// TIA Portal V20 export
FUNCTION "CollectAlarms" : Void   // FC64, LAD
TITLE = Alarm Collector Unit
AUTHOR : ERsystem_FA2_DH. Kim
// Collects alarms from the respective level and categorises the alarms into the different alarm classes.
// stored: Namespace Unit1, SetENOAutomatically false
   VAR_INPUT
      resetAlarms : Bool;
      disableAlarms : Bool;
   END_VAR
   VAR_OUTPUT
      commandsToUnit : "LUC_typeStateCommands";   // Feedback to the unit
   END_VAR
   VAR CONSTANT
      DelayTime : Time := T#300ms;
      TRUE : Bool := TRUE;
      FALSE : Bool;
   END_VAR
BEGIN

REGION Network 1: Reset Alarms
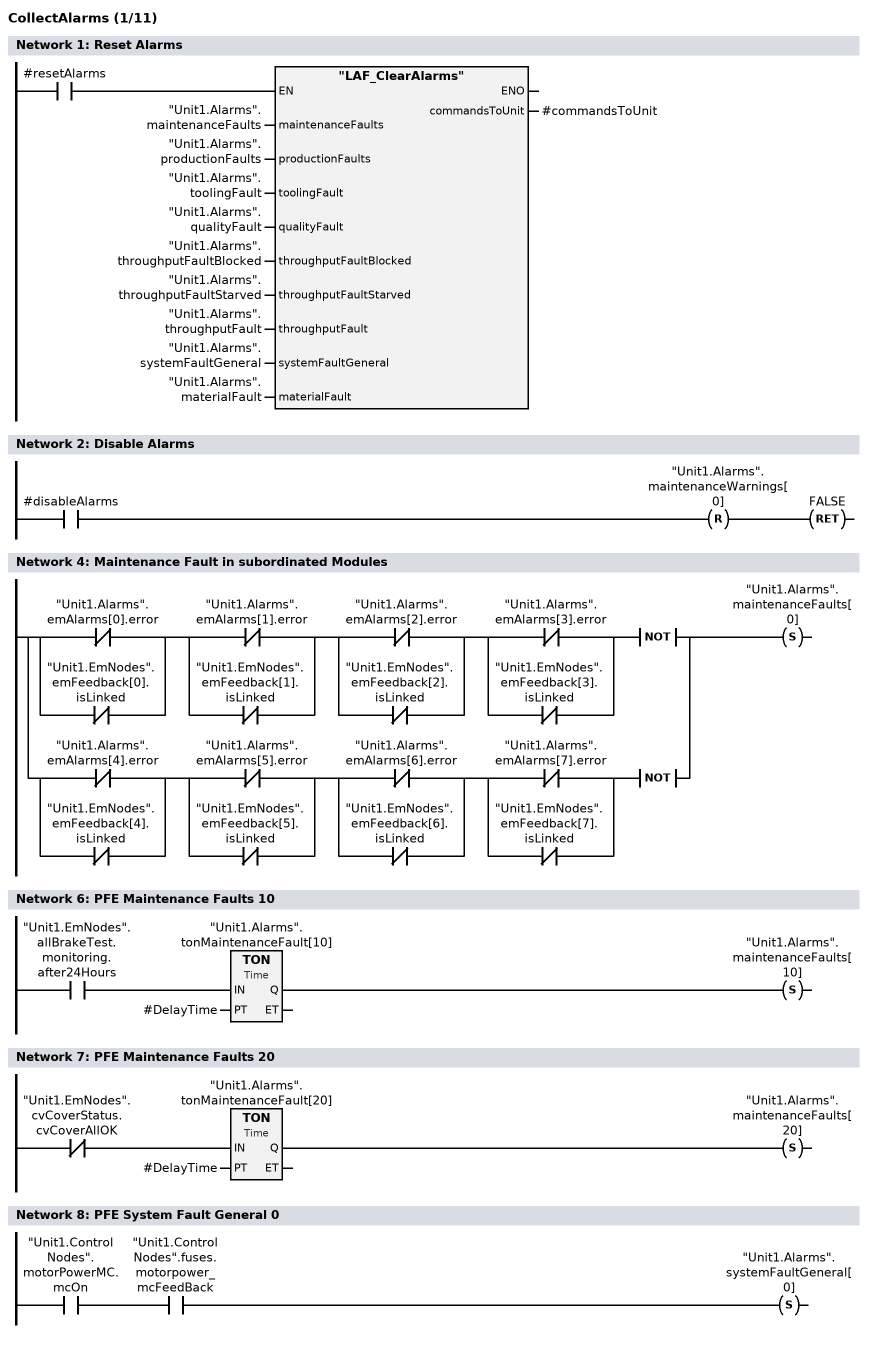
   RUNG wire#powerrail
      Contact( #resetAlarms )
      "LAF_ClearAlarms"(maintenanceFaults := "Unit1.Alarms".maintenanceFaults, productionFaults := "Unit1.Alarms".productionFaults, toolingFault := "Unit1.Alarms".toolingFault, qualityFault := "Unit1.Alarms".qualityFault, throughputFaultBlocked := "Unit1.Alarms".throughputFaultBlocked, throughputFaultStarved := "Unit1.Alarms".throughputFaultStarved, throughputFault := "Unit1.Alarms".throughputFault, systemFaultGeneral := "Unit1.Alarms".systemFaultGeneral, materialFault := "Unit1.Alarms".materialFault, commandsToUnit => #commandsToUnit)
   END_RUNG
   // the same network as SCL:
   IF #resetAlarms THEN
       "LAF_ClearAlarms"(maintenanceFaults := "Unit1.Alarms".maintenanceFaults,
                         productionFaults := "Unit1.Alarms".productionFaults,
                         toolingFault := "Unit1.Alarms".toolingFault,
                         qualityFault := "Unit1.Alarms".qualityFault,
                         throughputFaultBlocked := "Unit1.Alarms".throughputFaultBlocked,
                         throughputFaultStarved := "Unit1.Alarms".throughputFaultStarved,
                         throughputFault := "Unit1.Alarms".throughputFault,
                         systemFaultGeneral := "Unit1.Alarms".systemFaultGeneral,
                         materialFault := "Unit1.Alarms".materialFault,
                         commandsToUnit => #commandsToUnit);
   END_IF;
END_REGION

REGION Network 2: Disable Alarms
   RUNG wire#powerrail
      Contact( #disableAlarms )
      R_Coil( "Unit1.Alarms".maintenanceWarnings[0] )
      ReturnCoil( FALSE )
   END_RUNG
   // the same network as SCL:
   IF #disableAlarms THEN
       "Unit1.Alarms".maintenanceWarnings[0] := FALSE;
       ENO := FALSE;
       RETURN;
   END_IF;
END_REGION

REGION Network 3: *************** Fault ************************
END_REGION

REGION Network 4: Maintenance Fault in subordinated Modules
   RUNG wire#powerrail
      I_Contact( "Unit1.Alarms".emAlarms[0].error )
      wire#w1
      I_Contact( "Unit1.Alarms".emAlarms[1].error )
      wire#w2
      I_Contact( "Unit1.Alarms".emAlarms[2].error )
      wire#w3
      I_Contact( "Unit1.Alarms".emAlarms[3].error )
      wire#w4
      Not()
      wire#w5
      S_Coil( "Unit1.Alarms".maintenanceFaults[0] )
   END_RUNG
   RUNG wire#powerrail
      I_Contact( "Unit1.EmNodes".emFeedback[0].isLinked )
   END_RUNG wire#w1
   RUNG wire#w1
      I_Contact( "Unit1.EmNodes".emFeedback[1].isLinked )
   END_RUNG wire#w2
   RUNG wire#w2
      I_Contact( "Unit1.EmNodes".emFeedback[2].isLinked )
   END_RUNG wire#w3
   RUNG wire#w3
      I_Contact( "Unit1.EmNodes".emFeedback[3].isLinked )
   END_RUNG wire#w4
   RUNG wire#powerrail
      I_Contact( "Unit1.Alarms".emAlarms[4].error )
      wire#w6
      I_Contact( "Unit1.Alarms".emAlarms[5].error )
      wire#w7
      I_Contact( "Unit1.Alarms".emAlarms[6].error )
      wire#w8
      I_Contact( "Unit1.Alarms".emAlarms[7].error )
      wire#w9
      Not()
   END_RUNG wire#w5
   RUNG wire#powerrail
      I_Contact( "Unit1.EmNodes".emFeedback[4].isLinked )
   END_RUNG wire#w6
   RUNG wire#w6
      I_Contact( "Unit1.EmNodes".emFeedback[5].isLinked )
   END_RUNG wire#w7
   RUNG wire#w7
      I_Contact( "Unit1.EmNodes".emFeedback[6].isLinked )
   END_RUNG wire#w8
   RUNG wire#w8
      I_Contact( "Unit1.EmNodes".emFeedback[7].isLinked )
   END_RUNG wire#w9
   // the same network as SCL:
   IF NOT ((NOT "Unit1.Alarms".emAlarms[0].error OR NOT "Unit1.EmNodes".emFeedback[0].isLinked) AND (NOT "Unit1.Alarms".emAlarms[1].error OR NOT "Unit1.EmNodes".emFeedback[1].isLinked) AND (NOT "Unit1.Alarms".emAlarms[2].error OR NOT "Unit1.EmNodes".emFeedback[2].isLinked) AND (NOT "Unit1.Alarms".emAlarms[3].error OR NOT "Unit1.EmNodes".emFeedback[3].isLinked)) OR NOT ((NOT "Unit1.Alarms".emAlarms[4].error OR NOT "Unit1.EmNodes".emFeedback[4].isLinked) AND (NOT "Unit1.Alarms".emAlarms[5].error OR NOT "Unit1.EmNodes".emFeedback[5].isLinked) AND (NOT "Unit1.Alarms".emAlarms[6].error OR NOT "Unit1.EmNodes".emFeedback[6].isLinked) AND (NOT "Unit1.Alarms".emAlarms[7].error OR NOT "Unit1.EmNodes".emFeedback[7].isLinked)) THEN
       "Unit1.Alarms".maintenanceFaults[0] := TRUE;
   END_IF;
END_REGION

REGION Network 5: PFE Maintenance Faults 1
END_REGION

REGION Network 6: PFE Maintenance Faults 10
   RUNG wire#powerrail
      Contact( "Unit1.EmNodes".allBrakeTest.monitoring.after24Hours )
      { S7_Templates := "time_type := Time" } "Unit1.Alarms".tonMaintenanceFault[10].TON(pt := #DelayTime, et =>)
      S_Coil( "Unit1.Alarms".maintenanceFaults[10] )
   END_RUNG
   // the same network as SCL:
   "Unit1.Alarms".tonMaintenanceFault[10].TON(IN := "Unit1.EmNodes".allBrakeTest.monitoring.after24Hours,
                           PT := #DelayTime);
   IF "Unit1.Alarms".tonMaintenanceFault[10].Q THEN "Unit1.Alarms".maintenanceFaults[10] := TRUE; END_IF;
END_REGION

REGION Network 7: PFE Maintenance Faults 20
   RUNG wire#powerrail
      I_Contact( "Unit1.EmNodes".cvCoverStatus.cvCoverAllOK )
      { S7_Templates := "time_type := Time" } "Unit1.Alarms".tonMaintenanceFault[20].TON(pt := #DelayTime, et =>)
      S_Coil( "Unit1.Alarms".maintenanceFaults[20] )
   END_RUNG
   // the same network as SCL:
   "Unit1.Alarms".tonMaintenanceFault[20].TON(IN := NOT "Unit1.EmNodes".cvCoverStatus.cvCoverAllOK,
                           PT := #DelayTime);
   IF "Unit1.Alarms".tonMaintenanceFault[20].Q THEN "Unit1.Alarms".maintenanceFaults[20] := TRUE; END_IF;
END_REGION

REGION Network 8: PFE System Fault General 0
   RUNG wire#powerrail
      Contact( "Unit1.ControlNodes".motorPowerMC.mcOn )
      Contact( "Unit1.ControlNodes".fuses.motorpower_mcFeedBack )
      S_Coil( "Unit1.Alarms".systemFaultGeneral[0] )
   END_RUNG
   // the same network as SCL:
   IF "Unit1.ControlNodes".motorPowerMC.mcOn AND "Unit1.ControlNodes".fuses.motorpower_mcFeedBack THEN
       "Unit1.Alarms".systemFaultGeneral[0] := TRUE;
   END_IF;
END_REGION

REGION Network 9: PFE System Fault General 1
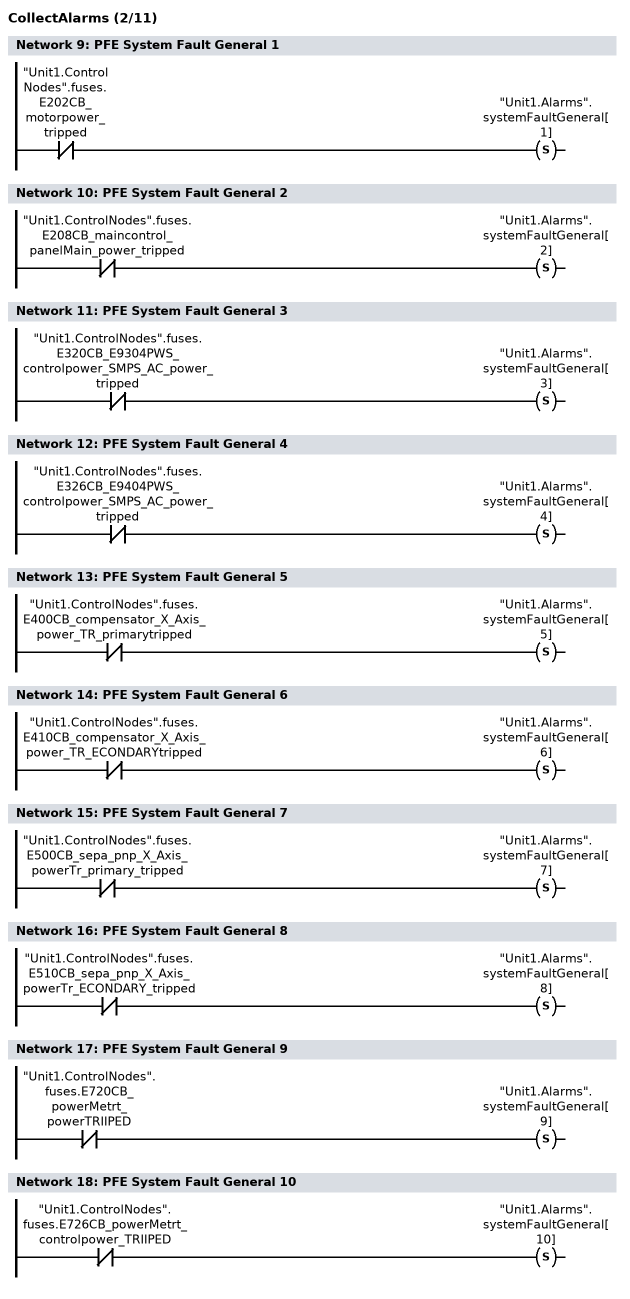
   RUNG wire#powerrail
      I_Contact( "Unit1.ControlNodes".fuses.E202CB_motorpower_tripped )
      S_Coil( "Unit1.Alarms".systemFaultGeneral[1] )
   END_RUNG
   // the same network as SCL:
   IF NOT "Unit1.ControlNodes".fuses.E202CB_motorpower_tripped THEN
       "Unit1.Alarms".systemFaultGeneral[1] := TRUE;
   END_IF;
END_REGION

REGION Network 10: PFE System Fault General 2
   RUNG wire#powerrail
      I_Contact( "Unit1.ControlNodes".fuses.E208CB_maincontrol_panelMain_power_tripped )
      S_Coil( "Unit1.Alarms".systemFaultGeneral[2] )
   END_RUNG
   // the same network as SCL:
   IF NOT "Unit1.ControlNodes".fuses.E208CB_maincontrol_panelMain_power_tripped THEN
       "Unit1.Alarms".systemFaultGeneral[2] := TRUE;
   END_IF;
END_REGION

REGION Network 11: PFE System Fault General 3
   RUNG wire#powerrail
      I_Contact( "Unit1.ControlNodes".fuses.E320CB_E9304PWS_controlpower_SMPS_AC_power_tripped )
      S_Coil( "Unit1.Alarms".systemFaultGeneral[3] )
   END_RUNG
   // the same network as SCL:
   IF NOT "Unit1.ControlNodes".fuses.E320CB_E9304PWS_controlpower_SMPS_AC_power_tripped THEN
       "Unit1.Alarms".systemFaultGeneral[3] := TRUE;
   END_IF;
END_REGION

REGION Network 12: PFE System Fault General 4
   RUNG wire#powerrail
      I_Contact( "Unit1.ControlNodes".fuses.E326CB_E9404PWS_controlpower_SMPS_AC_power_tripped )
      S_Coil( "Unit1.Alarms".systemFaultGeneral[4] )
   END_RUNG
   // the same network as SCL:
   IF NOT "Unit1.ControlNodes".fuses.E326CB_E9404PWS_controlpower_SMPS_AC_power_tripped THEN
       "Unit1.Alarms".systemFaultGeneral[4] := TRUE;
   END_IF;
END_REGION

REGION Network 13: PFE System Fault General 5
   RUNG wire#powerrail
      I_Contact( "Unit1.ControlNodes".fuses.E400CB_compensator_X_Axis_power_TR_primarytripped )
      S_Coil( "Unit1.Alarms".systemFaultGeneral[5] )
   END_RUNG
   // the same network as SCL:
   IF NOT "Unit1.ControlNodes".fuses.E400CB_compensator_X_Axis_power_TR_primarytripped THEN
       "Unit1.Alarms".systemFaultGeneral[5] := TRUE;
   END_IF;
END_REGION

REGION Network 14: PFE System Fault General 6
   RUNG wire#powerrail
      I_Contact( "Unit1.ControlNodes".fuses.E410CB_compensator_X_Axis_power_TR_ECONDARYtripped )
      S_Coil( "Unit1.Alarms".systemFaultGeneral[6] )
   END_RUNG
   // the same network as SCL:
   IF NOT "Unit1.ControlNodes".fuses.E410CB_compensator_X_Axis_power_TR_ECONDARYtripped THEN
       "Unit1.Alarms".systemFaultGeneral[6] := TRUE;
   END_IF;
END_REGION

REGION Network 15: PFE System Fault General 7
   RUNG wire#powerrail
      I_Contact( "Unit1.ControlNodes".fuses.E500CB_sepa_pnp_X_Axis_powerTr_primary_tripped )
      S_Coil( "Unit1.Alarms".systemFaultGeneral[7] )
   END_RUNG
   // the same network as SCL:
   IF NOT "Unit1.ControlNodes".fuses.E500CB_sepa_pnp_X_Axis_powerTr_primary_tripped THEN
       "Unit1.Alarms".systemFaultGeneral[7] := TRUE;
   END_IF;
END_REGION

REGION Network 16: PFE System Fault General 8
   RUNG wire#powerrail
      I_Contact( "Unit1.ControlNodes".fuses.E510CB_sepa_pnp_X_Axis_powerTr_ECONDARY_tripped )
      S_Coil( "Unit1.Alarms".systemFaultGeneral[8] )
   END_RUNG
   // the same network as SCL:
   IF NOT "Unit1.ControlNodes".fuses.E510CB_sepa_pnp_X_Axis_powerTr_ECONDARY_tripped THEN
       "Unit1.Alarms".systemFaultGeneral[8] := TRUE;
   END_IF;
END_REGION

REGION Network 17: PFE System Fault General 9
   RUNG wire#powerrail
      I_Contact( "Unit1.ControlNodes".fuses.E720CB_powerMetrt_powerTRIIPED )
      S_Coil( "Unit1.Alarms".systemFaultGeneral[9] )
   END_RUNG
   // the same network as SCL:
   IF NOT "Unit1.ControlNodes".fuses.E720CB_powerMetrt_powerTRIIPED THEN
       "Unit1.Alarms".systemFaultGeneral[9] := TRUE;
   END_IF;
END_REGION

REGION Network 18: PFE System Fault General 10
   RUNG wire#powerrail
      I_Contact( "Unit1.ControlNodes".fuses.E726CB_powerMetrt_controlpower_TRIIPED )
      S_Coil( "Unit1.Alarms".systemFaultGeneral[10] )
   END_RUNG
   // the same network as SCL:
   IF NOT "Unit1.ControlNodes".fuses.E726CB_powerMetrt_controlpower_TRIIPED THEN
       "Unit1.Alarms".systemFaultGeneral[10] := TRUE;
   END_IF;
END_REGION

REGION Network 19: PFE System Fault General 11
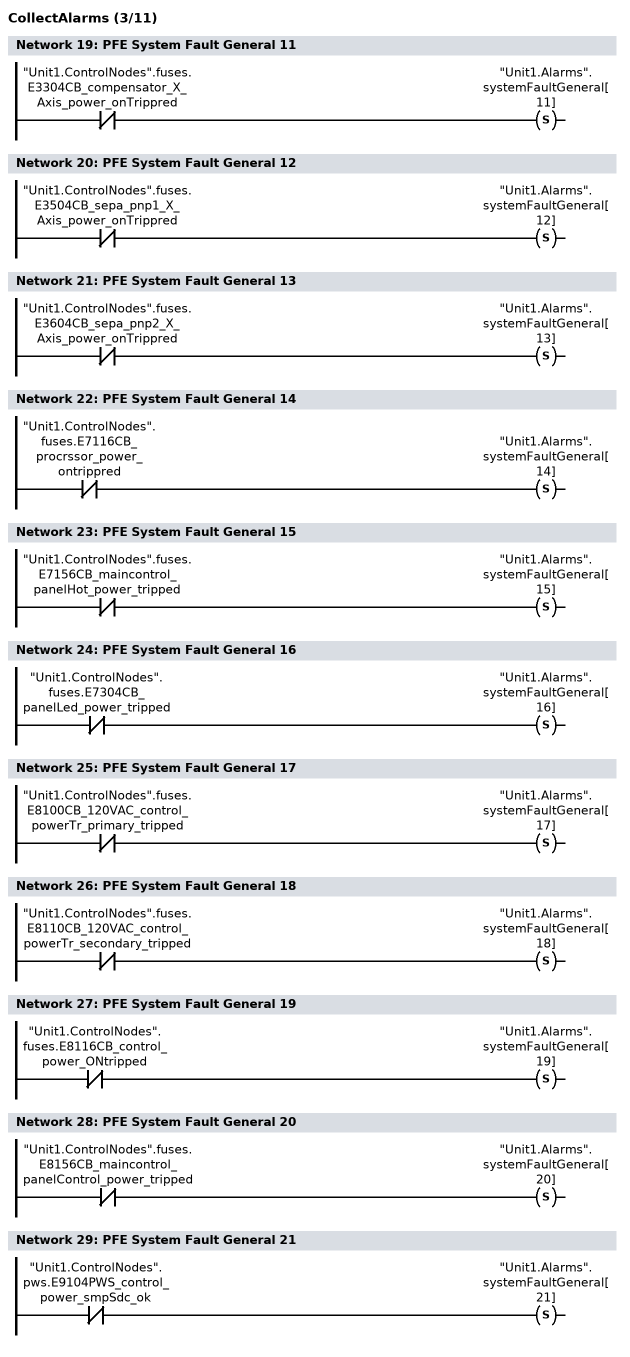
   RUNG wire#powerrail
      I_Contact( "Unit1.ControlNodes".fuses.E3304CB_compensator_X_Axis_power_onTrippred )
      S_Coil( "Unit1.Alarms".systemFaultGeneral[11] )
   END_RUNG
   // the same network as SCL:
   IF NOT "Unit1.ControlNodes".fuses.E3304CB_compensator_X_Axis_power_onTrippred THEN
       "Unit1.Alarms".systemFaultGeneral[11] := TRUE;
   END_IF;
END_REGION

REGION Network 20: PFE System Fault General 12
   RUNG wire#powerrail
      I_Contact( "Unit1.ControlNodes".fuses.E3504CB_sepa_pnp1_X_Axis_power_onTrippred )
      S_Coil( "Unit1.Alarms".systemFaultGeneral[12] )
   END_RUNG
   // the same network as SCL:
   IF NOT "Unit1.ControlNodes".fuses.E3504CB_sepa_pnp1_X_Axis_power_onTrippred THEN
       "Unit1.Alarms".systemFaultGeneral[12] := TRUE;
   END_IF;
END_REGION

REGION Network 21: PFE System Fault General 13
   RUNG wire#powerrail
      I_Contact( "Unit1.ControlNodes".fuses.E3604CB_sepa_pnp2_X_Axis_power_onTrippred )
      S_Coil( "Unit1.Alarms".systemFaultGeneral[13] )
   END_RUNG
   // the same network as SCL:
   IF NOT "Unit1.ControlNodes".fuses.E3604CB_sepa_pnp2_X_Axis_power_onTrippred THEN
       "Unit1.Alarms".systemFaultGeneral[13] := TRUE;
   END_IF;
END_REGION

REGION Network 22: PFE System Fault General 14
   RUNG wire#powerrail
      I_Contact( "Unit1.ControlNodes".fuses.E7116CB_procrssor_power_ontrippred )
      S_Coil( "Unit1.Alarms".systemFaultGeneral[14] )
   END_RUNG
   // the same network as SCL:
   IF NOT "Unit1.ControlNodes".fuses.E7116CB_procrssor_power_ontrippred THEN
       "Unit1.Alarms".systemFaultGeneral[14] := TRUE;
   END_IF;
END_REGION

REGION Network 23: PFE System Fault General 15
   RUNG wire#powerrail
      I_Contact( "Unit1.ControlNodes".fuses.E7156CB_maincontrol_panelHot_power_tripped )
      S_Coil( "Unit1.Alarms".systemFaultGeneral[15] )
   END_RUNG
   // the same network as SCL:
   IF NOT "Unit1.ControlNodes".fuses.E7156CB_maincontrol_panelHot_power_tripped THEN
       "Unit1.Alarms".systemFaultGeneral[15] := TRUE;
   END_IF;
END_REGION

REGION Network 24: PFE System Fault General 16
   RUNG wire#powerrail
      I_Contact( "Unit1.ControlNodes".fuses.E7304CB_panelLed_power_tripped )
      S_Coil( "Unit1.Alarms".systemFaultGeneral[16] )
   END_RUNG
   // the same network as SCL:
   IF NOT "Unit1.ControlNodes".fuses.E7304CB_panelLed_power_tripped THEN
       "Unit1.Alarms".systemFaultGeneral[16] := TRUE;
   END_IF;
END_REGION

REGION Network 25: PFE System Fault General 17
   RUNG wire#powerrail
      I_Contact( "Unit1.ControlNodes".fuses.E8100CB_120VAC_control_powerTr_primary_tripped )
      S_Coil( "Unit1.Alarms".systemFaultGeneral[17] )
   END_RUNG
   // the same network as SCL:
   IF NOT "Unit1.ControlNodes".fuses.E8100CB_120VAC_control_powerTr_primary_tripped THEN
       "Unit1.Alarms".systemFaultGeneral[17] := TRUE;
   END_IF;
END_REGION

REGION Network 26: PFE System Fault General 18
   RUNG wire#powerrail
      I_Contact( "Unit1.ControlNodes".fuses.E8110CB_120VAC_control_powerTr_secondary_tripped )
      S_Coil( "Unit1.Alarms".systemFaultGeneral[18] )
   END_RUNG
   // the same network as SCL:
   IF NOT "Unit1.ControlNodes".fuses.E8110CB_120VAC_control_powerTr_secondary_tripped THEN
       "Unit1.Alarms".systemFaultGeneral[18] := TRUE;
   END_IF;
END_REGION

REGION Network 27: PFE System Fault General 19
   RUNG wire#powerrail
      I_Contact( "Unit1.ControlNodes".fuses.E8116CB_control_power_ONtripped )
      S_Coil( "Unit1.Alarms".systemFaultGeneral[19] )
   END_RUNG
   // the same network as SCL:
   IF NOT "Unit1.ControlNodes".fuses.E8116CB_control_power_ONtripped THEN
       "Unit1.Alarms".systemFaultGeneral[19] := TRUE;
   END_IF;
END_REGION

REGION Network 28: PFE System Fault General 20
   RUNG wire#powerrail
      I_Contact( "Unit1.ControlNodes".fuses.E8156CB_maincontrol_panelControl_power_tripped )
      S_Coil( "Unit1.Alarms".systemFaultGeneral[20] )
   END_RUNG
   // the same network as SCL:
   IF NOT "Unit1.ControlNodes".fuses.E8156CB_maincontrol_panelControl_power_tripped THEN
       "Unit1.Alarms".systemFaultGeneral[20] := TRUE;
   END_IF;
END_REGION

REGION Network 29: PFE System Fault General 21
   RUNG wire#powerrail
      I_Contact( "Unit1.ControlNodes".pws.E9104PWS_control_power_smpSdc_ok )
      S_Coil( "Unit1.Alarms".systemFaultGeneral[21] )
   END_RUNG
   // the same network as SCL:
   IF NOT "Unit1.ControlNodes".pws.E9104PWS_control_power_smpSdc_ok THEN
       "Unit1.Alarms".systemFaultGeneral[21] := TRUE;
   END_IF;
END_REGION

REGION Network 30: PFE System Fault General 22
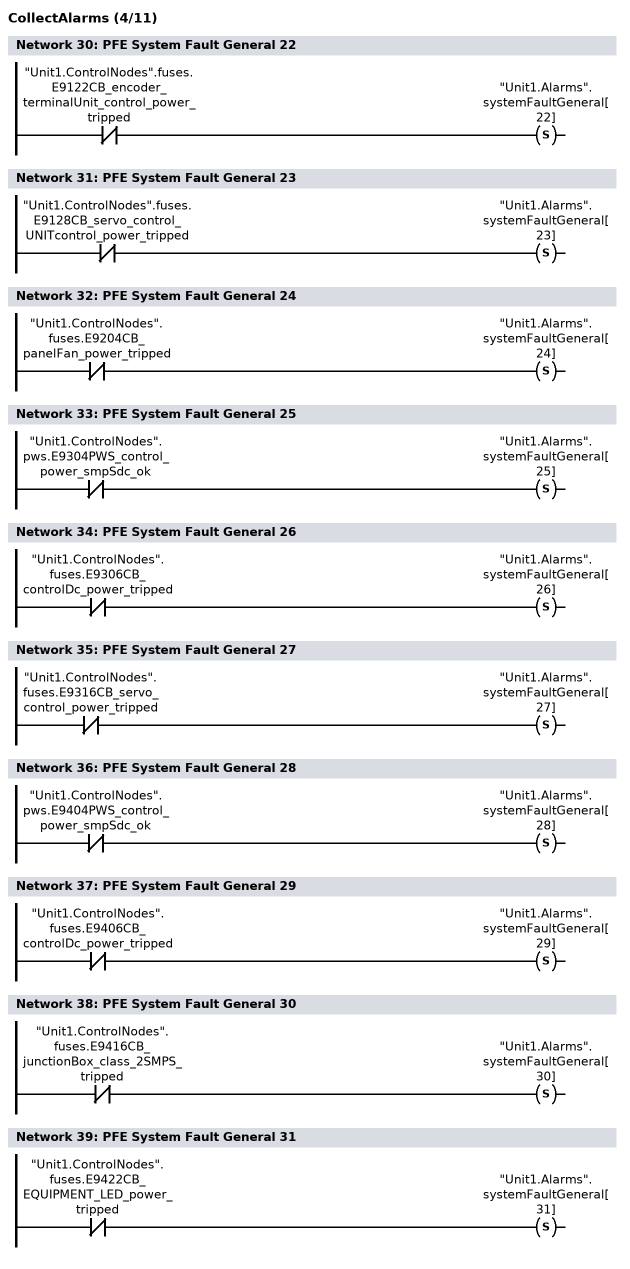
   RUNG wire#powerrail
      I_Contact( "Unit1.ControlNodes".fuses.E9122CB_encoder_terminalUnit_control_power_tripped )
      S_Coil( "Unit1.Alarms".systemFaultGeneral[22] )
   END_RUNG
   // the same network as SCL:
   IF NOT "Unit1.ControlNodes".fuses.E9122CB_encoder_terminalUnit_control_power_tripped THEN
       "Unit1.Alarms".systemFaultGeneral[22] := TRUE;
   END_IF;
END_REGION

REGION Network 31: PFE System Fault General 23
   RUNG wire#powerrail
      I_Contact( "Unit1.ControlNodes".fuses.E9128CB_servo_control_UNITcontrol_power_tripped )
      S_Coil( "Unit1.Alarms".systemFaultGeneral[23] )
   END_RUNG
   // the same network as SCL:
   IF NOT "Unit1.ControlNodes".fuses.E9128CB_servo_control_UNITcontrol_power_tripped THEN
       "Unit1.Alarms".systemFaultGeneral[23] := TRUE;
   END_IF;
END_REGION

REGION Network 32: PFE System Fault General 24
   RUNG wire#powerrail
      I_Contact( "Unit1.ControlNodes".fuses.E9204CB_panelFan_power_tripped )
      S_Coil( "Unit1.Alarms".systemFaultGeneral[24] )
   END_RUNG
   // the same network as SCL:
   IF NOT "Unit1.ControlNodes".fuses.E9204CB_panelFan_power_tripped THEN
       "Unit1.Alarms".systemFaultGeneral[24] := TRUE;
   END_IF;
END_REGION

REGION Network 33: PFE System Fault General 25
   RUNG wire#powerrail
      I_Contact( "Unit1.ControlNodes".pws.E9304PWS_control_power_smpSdc_ok )
      S_Coil( "Unit1.Alarms".systemFaultGeneral[25] )
   END_RUNG
   // the same network as SCL:
   IF NOT "Unit1.ControlNodes".pws.E9304PWS_control_power_smpSdc_ok THEN
       "Unit1.Alarms".systemFaultGeneral[25] := TRUE;
   END_IF;
END_REGION

REGION Network 34: PFE System Fault General 26
   RUNG wire#powerrail
      I_Contact( "Unit1.ControlNodes".fuses.E9306CB_controlDc_power_tripped )
      S_Coil( "Unit1.Alarms".systemFaultGeneral[26] )
   END_RUNG
   // the same network as SCL:
   IF NOT "Unit1.ControlNodes".fuses.E9306CB_controlDc_power_tripped THEN
       "Unit1.Alarms".systemFaultGeneral[26] := TRUE;
   END_IF;
END_REGION

REGION Network 35: PFE System Fault General 27
   RUNG wire#powerrail
      I_Contact( "Unit1.ControlNodes".fuses.E9316CB_servo_control_power_tripped )
      S_Coil( "Unit1.Alarms".systemFaultGeneral[27] )
   END_RUNG
   // the same network as SCL:
   IF NOT "Unit1.ControlNodes".fuses.E9316CB_servo_control_power_tripped THEN
       "Unit1.Alarms".systemFaultGeneral[27] := TRUE;
   END_IF;
END_REGION

REGION Network 36: PFE System Fault General 28
   RUNG wire#powerrail
      I_Contact( "Unit1.ControlNodes".pws.E9404PWS_control_power_smpSdc_ok )
      S_Coil( "Unit1.Alarms".systemFaultGeneral[28] )
   END_RUNG
   // the same network as SCL:
   IF NOT "Unit1.ControlNodes".pws.E9404PWS_control_power_smpSdc_ok THEN
       "Unit1.Alarms".systemFaultGeneral[28] := TRUE;
   END_IF;
END_REGION

REGION Network 37: PFE System Fault General 29
   RUNG wire#powerrail
      I_Contact( "Unit1.ControlNodes".fuses.E9406CB_controlDc_power_tripped )
      S_Coil( "Unit1.Alarms".systemFaultGeneral[29] )
   END_RUNG
   // the same network as SCL:
   IF NOT "Unit1.ControlNodes".fuses.E9406CB_controlDc_power_tripped THEN
       "Unit1.Alarms".systemFaultGeneral[29] := TRUE;
   END_IF;
END_REGION

REGION Network 38: PFE System Fault General 30
   RUNG wire#powerrail
      I_Contact( "Unit1.ControlNodes".fuses.E9416CB_junctionBox_class_2SMPS_tripped )
      S_Coil( "Unit1.Alarms".systemFaultGeneral[30] )
   END_RUNG
   // the same network as SCL:
   IF NOT "Unit1.ControlNodes".fuses.E9416CB_junctionBox_class_2SMPS_tripped THEN
       "Unit1.Alarms".systemFaultGeneral[30] := TRUE;
   END_IF;
END_REGION

REGION Network 39: PFE System Fault General 31
   RUNG wire#powerrail
      I_Contact( "Unit1.ControlNodes".fuses.E9422CB_EQUIPMENT_LED_power_tripped )
      S_Coil( "Unit1.Alarms".systemFaultGeneral[31] )
   END_RUNG
   // the same network as SCL:
   IF NOT "Unit1.ControlNodes".fuses.E9422CB_EQUIPMENT_LED_power_tripped THEN
       "Unit1.Alarms".systemFaultGeneral[31] := TRUE;
   END_IF;
END_REGION

REGION Network 40: PFE System Fault General 32
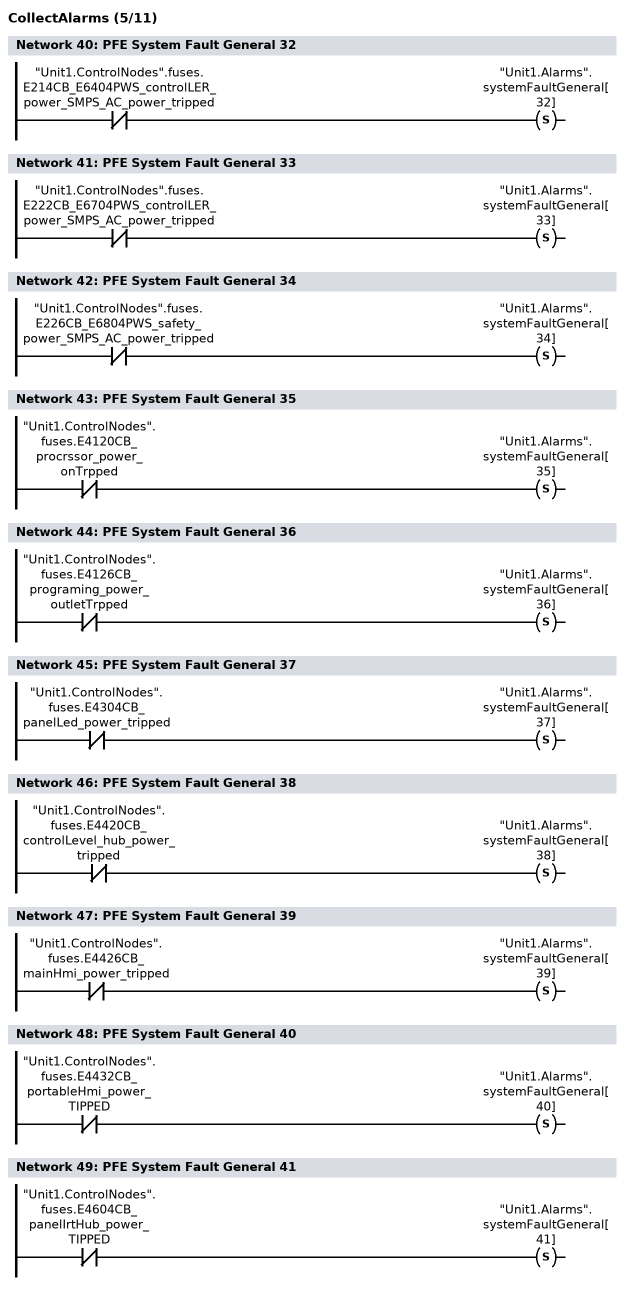
   RUNG wire#powerrail
      I_Contact( "Unit1.ControlNodes".fuses.E214CB_E6404PWS_controlLER_power_SMPS_AC_power_tripped )
      S_Coil( "Unit1.Alarms".systemFaultGeneral[32] )
   END_RUNG
   // the same network as SCL:
   IF NOT "Unit1.ControlNodes".fuses.E214CB_E6404PWS_controlLER_power_SMPS_AC_power_tripped THEN
       "Unit1.Alarms".systemFaultGeneral[32] := TRUE;
   END_IF;
END_REGION

REGION Network 41: PFE System Fault General 33
   RUNG wire#powerrail
      I_Contact( "Unit1.ControlNodes".fuses.E222CB_E6704PWS_controlLER_power_SMPS_AC_power_tripped )
      S_Coil( "Unit1.Alarms".systemFaultGeneral[33] )
   END_RUNG
   // the same network as SCL:
   IF NOT "Unit1.ControlNodes".fuses.E222CB_E6704PWS_controlLER_power_SMPS_AC_power_tripped THEN
       "Unit1.Alarms".systemFaultGeneral[33] := TRUE;
   END_IF;
END_REGION

REGION Network 42: PFE System Fault General 34
   RUNG wire#powerrail
      I_Contact( "Unit1.ControlNodes".fuses.E226CB_E6804PWS_safety_power_SMPS_AC_power_tripped )
      S_Coil( "Unit1.Alarms".systemFaultGeneral[34] )
   END_RUNG
   // the same network as SCL:
   IF NOT "Unit1.ControlNodes".fuses.E226CB_E6804PWS_safety_power_SMPS_AC_power_tripped THEN
       "Unit1.Alarms".systemFaultGeneral[34] := TRUE;
   END_IF;
END_REGION

REGION Network 43: PFE System Fault General 35
   RUNG wire#powerrail
      I_Contact( "Unit1.ControlNodes".fuses.E4120CB_procrssor_power_onTrpped )
      S_Coil( "Unit1.Alarms".systemFaultGeneral[35] )
   END_RUNG
   // the same network as SCL:
   IF NOT "Unit1.ControlNodes".fuses.E4120CB_procrssor_power_onTrpped THEN
       "Unit1.Alarms".systemFaultGeneral[35] := TRUE;
   END_IF;
END_REGION

REGION Network 44: PFE System Fault General 36
   RUNG wire#powerrail
      I_Contact( "Unit1.ControlNodes".fuses.E4126CB_programing_power_outletTrpped )
      S_Coil( "Unit1.Alarms".systemFaultGeneral[36] )
   END_RUNG
   // the same network as SCL:
   IF NOT "Unit1.ControlNodes".fuses.E4126CB_programing_power_outletTrpped THEN
       "Unit1.Alarms".systemFaultGeneral[36] := TRUE;
   END_IF;
END_REGION

REGION Network 45: PFE System Fault General 37
   RUNG wire#powerrail
      I_Contact( "Unit1.ControlNodes".fuses.E4304CB_panelLed_power_tripped )
      S_Coil( "Unit1.Alarms".systemFaultGeneral[37] )
   END_RUNG
   // the same network as SCL:
   IF NOT "Unit1.ControlNodes".fuses.E4304CB_panelLed_power_tripped THEN
       "Unit1.Alarms".systemFaultGeneral[37] := TRUE;
   END_IF;
END_REGION

REGION Network 46: PFE System Fault General 38
   RUNG wire#powerrail
      I_Contact( "Unit1.ControlNodes".fuses.E4420CB_controlLevel_hub_power_tripped )
      S_Coil( "Unit1.Alarms".systemFaultGeneral[38] )
   END_RUNG
   // the same network as SCL:
   IF NOT "Unit1.ControlNodes".fuses.E4420CB_controlLevel_hub_power_tripped THEN
       "Unit1.Alarms".systemFaultGeneral[38] := TRUE;
   END_IF;
END_REGION

REGION Network 47: PFE System Fault General 39
   RUNG wire#powerrail
      I_Contact( "Unit1.ControlNodes".fuses.E4426CB_mainHmi_power_tripped )
      S_Coil( "Unit1.Alarms".systemFaultGeneral[39] )
   END_RUNG
   // the same network as SCL:
   IF NOT "Unit1.ControlNodes".fuses.E4426CB_mainHmi_power_tripped THEN
       "Unit1.Alarms".systemFaultGeneral[39] := TRUE;
   END_IF;
END_REGION

REGION Network 48: PFE System Fault General 40
   RUNG wire#powerrail
      I_Contact( "Unit1.ControlNodes".fuses.E4432CB_portableHmi_power_TIPPED )
      S_Coil( "Unit1.Alarms".systemFaultGeneral[40] )
   END_RUNG
   // the same network as SCL:
   IF NOT "Unit1.ControlNodes".fuses.E4432CB_portableHmi_power_TIPPED THEN
       "Unit1.Alarms".systemFaultGeneral[40] := TRUE;
   END_IF;
END_REGION

REGION Network 49: PFE System Fault General 41
   RUNG wire#powerrail
      I_Contact( "Unit1.ControlNodes".fuses.E4604CB_panelIrtHub_power_TIPPED )
      S_Coil( "Unit1.Alarms".systemFaultGeneral[41] )
   END_RUNG
   // the same network as SCL:
   IF NOT "Unit1.ControlNodes".fuses.E4604CB_panelIrtHub_power_TIPPED THEN
       "Unit1.Alarms".systemFaultGeneral[41] := TRUE;
   END_IF;
END_REGION

REGION Network 50: PFE System Fault General 42
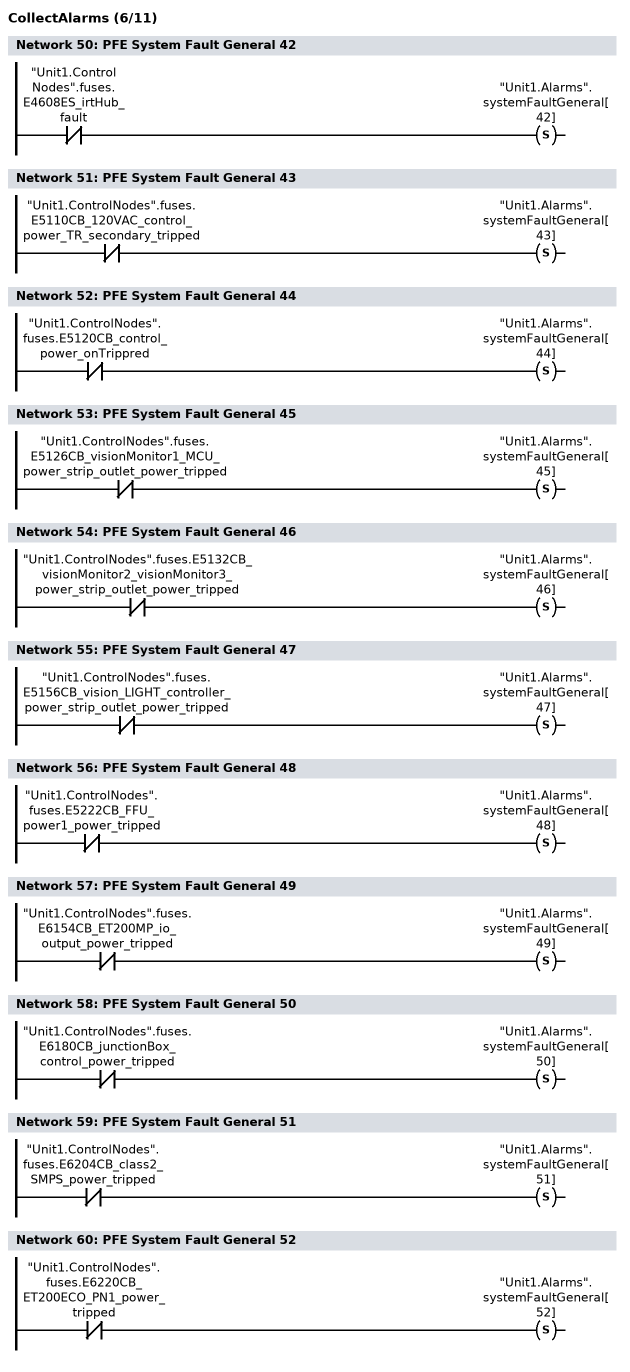
   RUNG wire#powerrail
      I_Contact( "Unit1.ControlNodes".fuses.E4608ES_irtHub_fault )
      S_Coil( "Unit1.Alarms".systemFaultGeneral[42] )
   END_RUNG
   // the same network as SCL:
   IF NOT "Unit1.ControlNodes".fuses.E4608ES_irtHub_fault THEN
       "Unit1.Alarms".systemFaultGeneral[42] := TRUE;
   END_IF;
END_REGION

REGION Network 51: PFE System Fault General 43
   RUNG wire#powerrail
      I_Contact( "Unit1.ControlNodes".fuses.E5110CB_120VAC_control_power_TR_secondary_tripped )
      S_Coil( "Unit1.Alarms".systemFaultGeneral[43] )
   END_RUNG
   // the same network as SCL:
   IF NOT "Unit1.ControlNodes".fuses.E5110CB_120VAC_control_power_TR_secondary_tripped THEN
       "Unit1.Alarms".systemFaultGeneral[43] := TRUE;
   END_IF;
END_REGION

REGION Network 52: PFE System Fault General 44
   RUNG wire#powerrail
      I_Contact( "Unit1.ControlNodes".fuses.E5120CB_control_power_onTrippred )
      S_Coil( "Unit1.Alarms".systemFaultGeneral[44] )
   END_RUNG
   // the same network as SCL:
   IF NOT "Unit1.ControlNodes".fuses.E5120CB_control_power_onTrippred THEN
       "Unit1.Alarms".systemFaultGeneral[44] := TRUE;
   END_IF;
END_REGION

REGION Network 53: PFE System Fault General 45
   RUNG wire#powerrail
      I_Contact( "Unit1.ControlNodes".fuses.E5126CB_visionMonitor1_MCU_power_strip_outlet_power_tripped )
      S_Coil( "Unit1.Alarms".systemFaultGeneral[45] )
   END_RUNG
   // the same network as SCL:
   IF NOT "Unit1.ControlNodes".fuses.E5126CB_visionMonitor1_MCU_power_strip_outlet_power_tripped THEN
       "Unit1.Alarms".systemFaultGeneral[45] := TRUE;
   END_IF;
END_REGION

REGION Network 54: PFE System Fault General 46
   RUNG wire#powerrail
      I_Contact( "Unit1.ControlNodes".fuses.E5132CB_visionMonitor2_visionMonitor3_power_strip_outlet_power_tripped )
      S_Coil( "Unit1.Alarms".systemFaultGeneral[46] )
   END_RUNG
   // the same network as SCL:
   IF NOT "Unit1.ControlNodes".fuses.E5132CB_visionMonitor2_visionMonitor3_power_strip_outlet_power_tripped THEN
       "Unit1.Alarms".systemFaultGeneral[46] := TRUE;
   END_IF;
END_REGION

REGION Network 55: PFE System Fault General 47
   RUNG wire#powerrail
      I_Contact( "Unit1.ControlNodes".fuses.E5156CB_vision_LIGHT_controller_power_strip_outlet_power_tripped )
      S_Coil( "Unit1.Alarms".systemFaultGeneral[47] )
   END_RUNG
   // the same network as SCL:
   IF NOT "Unit1.ControlNodes".fuses.E5156CB_vision_LIGHT_controller_power_strip_outlet_power_tripped THEN
       "Unit1.Alarms".systemFaultGeneral[47] := TRUE;
   END_IF;
END_REGION

REGION Network 56: PFE System Fault General 48
   RUNG wire#powerrail
      I_Contact( "Unit1.ControlNodes".fuses.E5222CB_FFU_power1_power_tripped )
      S_Coil( "Unit1.Alarms".systemFaultGeneral[48] )
   END_RUNG
   // the same network as SCL:
   IF NOT "Unit1.ControlNodes".fuses.E5222CB_FFU_power1_power_tripped THEN
       "Unit1.Alarms".systemFaultGeneral[48] := TRUE;
   END_IF;
END_REGION

REGION Network 57: PFE System Fault General 49
   RUNG wire#powerrail
      I_Contact( "Unit1.ControlNodes".fuses.E6154CB_ET200MP_io_output_power_tripped )
      S_Coil( "Unit1.Alarms".systemFaultGeneral[49] )
   END_RUNG
   // the same network as SCL:
   IF NOT "Unit1.ControlNodes".fuses.E6154CB_ET200MP_io_output_power_tripped THEN
       "Unit1.Alarms".systemFaultGeneral[49] := TRUE;
   END_IF;
END_REGION

REGION Network 58: PFE System Fault General 50
   RUNG wire#powerrail
      I_Contact( "Unit1.ControlNodes".fuses.E6180CB_junctionBox_control_power_tripped )
      S_Coil( "Unit1.Alarms".systemFaultGeneral[50] )
   END_RUNG
   // the same network as SCL:
   IF NOT "Unit1.ControlNodes".fuses.E6180CB_junctionBox_control_power_tripped THEN
       "Unit1.Alarms".systemFaultGeneral[50] := TRUE;
   END_IF;
END_REGION

REGION Network 59: PFE System Fault General 51
   RUNG wire#powerrail
      I_Contact( "Unit1.ControlNodes".fuses.E6204CB_class2_SMPS_power_tripped )
      S_Coil( "Unit1.Alarms".systemFaultGeneral[51] )
   END_RUNG
   // the same network as SCL:
   IF NOT "Unit1.ControlNodes".fuses.E6204CB_class2_SMPS_power_tripped THEN
       "Unit1.Alarms".systemFaultGeneral[51] := TRUE;
   END_IF;
END_REGION

REGION Network 60: PFE System Fault General 52
   RUNG wire#powerrail
      I_Contact( "Unit1.ControlNodes".fuses.E6220CB_ET200ECO_PN1_power_tripped )
      S_Coil( "Unit1.Alarms".systemFaultGeneral[52] )
   END_RUNG
   // the same network as SCL:
   IF NOT "Unit1.ControlNodes".fuses.E6220CB_ET200ECO_PN1_power_tripped THEN
       "Unit1.Alarms".systemFaultGeneral[52] := TRUE;
   END_IF;
END_REGION

REGION Network 61: PFE System Fault General 53
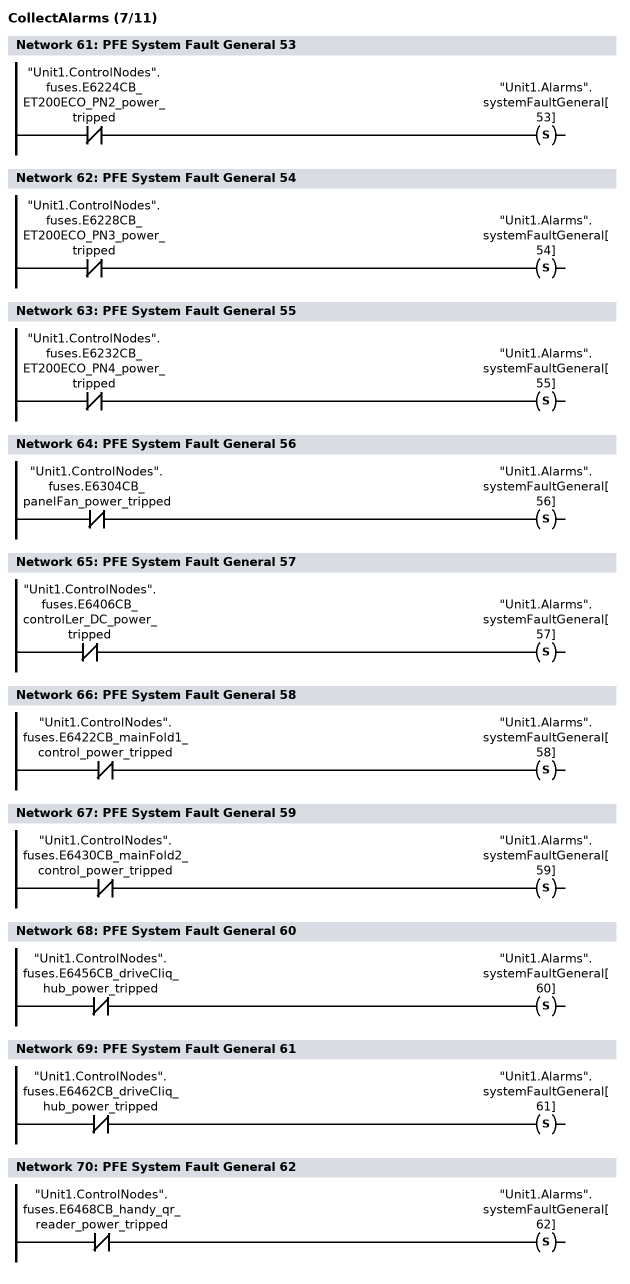
   RUNG wire#powerrail
      I_Contact( "Unit1.ControlNodes".fuses.E6224CB_ET200ECO_PN2_power_tripped )
      S_Coil( "Unit1.Alarms".systemFaultGeneral[53] )
   END_RUNG
   // the same network as SCL:
   IF NOT "Unit1.ControlNodes".fuses.E6224CB_ET200ECO_PN2_power_tripped THEN
       "Unit1.Alarms".systemFaultGeneral[53] := TRUE;
   END_IF;
END_REGION

REGION Network 62: PFE System Fault General 54
   RUNG wire#powerrail
      I_Contact( "Unit1.ControlNodes".fuses.E6228CB_ET200ECO_PN3_power_tripped )
      S_Coil( "Unit1.Alarms".systemFaultGeneral[54] )
   END_RUNG
   // the same network as SCL:
   IF NOT "Unit1.ControlNodes".fuses.E6228CB_ET200ECO_PN3_power_tripped THEN
       "Unit1.Alarms".systemFaultGeneral[54] := TRUE;
   END_IF;
END_REGION

REGION Network 63: PFE System Fault General 55
   RUNG wire#powerrail
      I_Contact( "Unit1.ControlNodes".fuses.E6232CB_ET200ECO_PN4_power_tripped )
      S_Coil( "Unit1.Alarms".systemFaultGeneral[55] )
   END_RUNG
   // the same network as SCL:
   IF NOT "Unit1.ControlNodes".fuses.E6232CB_ET200ECO_PN4_power_tripped THEN
       "Unit1.Alarms".systemFaultGeneral[55] := TRUE;
   END_IF;
END_REGION

REGION Network 64: PFE System Fault General 56
   RUNG wire#powerrail
      I_Contact( "Unit1.ControlNodes".fuses.E6304CB_panelFan_power_tripped )
      S_Coil( "Unit1.Alarms".systemFaultGeneral[56] )
   END_RUNG
   // the same network as SCL:
   IF NOT "Unit1.ControlNodes".fuses.E6304CB_panelFan_power_tripped THEN
       "Unit1.Alarms".systemFaultGeneral[56] := TRUE;
   END_IF;
END_REGION

REGION Network 65: PFE System Fault General 57
   RUNG wire#powerrail
      I_Contact( "Unit1.ControlNodes".fuses.E6406CB_controlLer_DC_power_tripped )
      S_Coil( "Unit1.Alarms".systemFaultGeneral[57] )
   END_RUNG
   // the same network as SCL:
   IF NOT "Unit1.ControlNodes".fuses.E6406CB_controlLer_DC_power_tripped THEN
       "Unit1.Alarms".systemFaultGeneral[57] := TRUE;
   END_IF;
END_REGION

REGION Network 66: PFE System Fault General 58
   RUNG wire#powerrail
      I_Contact( "Unit1.ControlNodes".fuses.E6422CB_mainFold1_control_power_tripped )
      S_Coil( "Unit1.Alarms".systemFaultGeneral[58] )
   END_RUNG
   // the same network as SCL:
   IF NOT "Unit1.ControlNodes".fuses.E6422CB_mainFold1_control_power_tripped THEN
       "Unit1.Alarms".systemFaultGeneral[58] := TRUE;
   END_IF;
END_REGION

REGION Network 67: PFE System Fault General 59
   RUNG wire#powerrail
      I_Contact( "Unit1.ControlNodes".fuses.E6430CB_mainFold2_control_power_tripped )
      S_Coil( "Unit1.Alarms".systemFaultGeneral[59] )
   END_RUNG
   // the same network as SCL:
   IF NOT "Unit1.ControlNodes".fuses.E6430CB_mainFold2_control_power_tripped THEN
       "Unit1.Alarms".systemFaultGeneral[59] := TRUE;
   END_IF;
END_REGION

REGION Network 68: PFE System Fault General 60
   RUNG wire#powerrail
      I_Contact( "Unit1.ControlNodes".fuses.E6456CB_driveCliq_hub_power_tripped )
      S_Coil( "Unit1.Alarms".systemFaultGeneral[60] )
   END_RUNG
   // the same network as SCL:
   IF NOT "Unit1.ControlNodes".fuses.E6456CB_driveCliq_hub_power_tripped THEN
       "Unit1.Alarms".systemFaultGeneral[60] := TRUE;
   END_IF;
END_REGION

REGION Network 69: PFE System Fault General 61
   RUNG wire#powerrail
      I_Contact( "Unit1.ControlNodes".fuses.E6462CB_driveCliq_hub_power_tripped )
      S_Coil( "Unit1.Alarms".systemFaultGeneral[61] )
   END_RUNG
   // the same network as SCL:
   IF NOT "Unit1.ControlNodes".fuses.E6462CB_driveCliq_hub_power_tripped THEN
       "Unit1.Alarms".systemFaultGeneral[61] := TRUE;
   END_IF;
END_REGION

REGION Network 70: PFE System Fault General 62
   RUNG wire#powerrail
      I_Contact( "Unit1.ControlNodes".fuses.E6468CB_handy_qr_reader_power_tripped )
      S_Coil( "Unit1.Alarms".systemFaultGeneral[62] )
   END_RUNG
   // the same network as SCL:
   IF NOT "Unit1.ControlNodes".fuses.E6468CB_handy_qr_reader_power_tripped THEN
       "Unit1.Alarms".systemFaultGeneral[62] := TRUE;
   END_IF;
END_REGION

REGION Network 71: PFE System Fault General 63
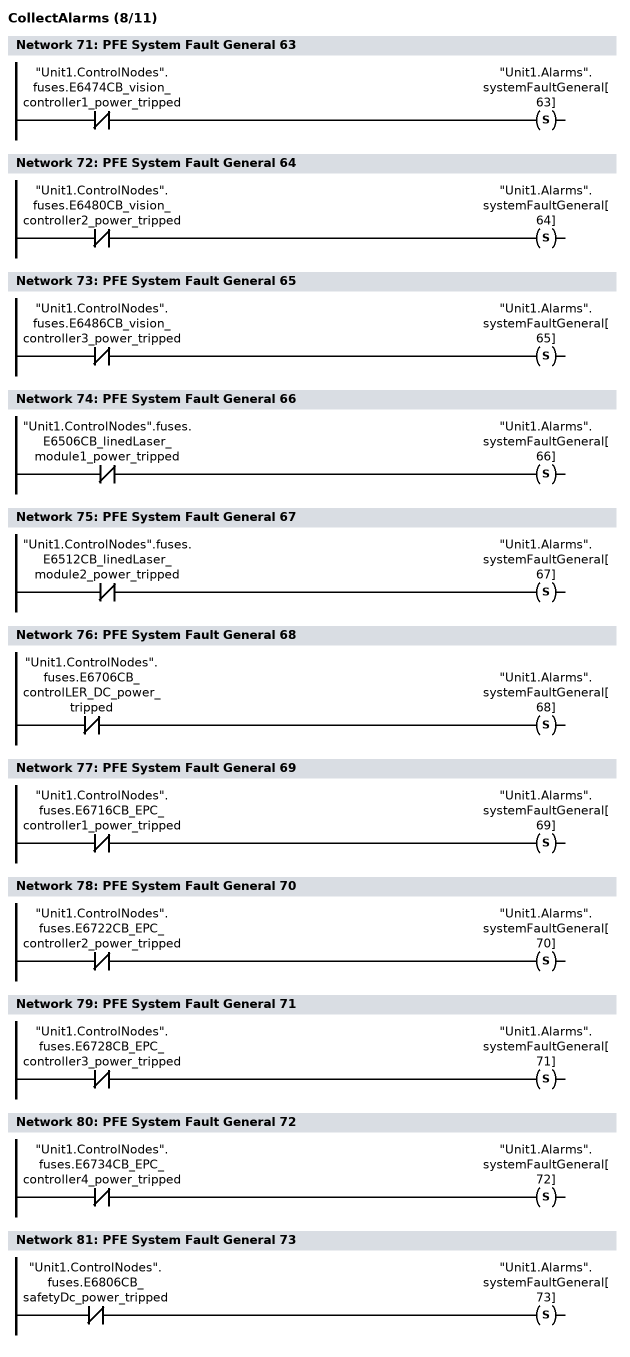
   RUNG wire#powerrail
      I_Contact( "Unit1.ControlNodes".fuses.E6474CB_vision_controller1_power_tripped )
      S_Coil( "Unit1.Alarms".systemFaultGeneral[63] )
   END_RUNG
   // the same network as SCL:
   IF NOT "Unit1.ControlNodes".fuses.E6474CB_vision_controller1_power_tripped THEN
       "Unit1.Alarms".systemFaultGeneral[63] := TRUE;
   END_IF;
END_REGION

REGION Network 72: PFE System Fault General 64
   RUNG wire#powerrail
      I_Contact( "Unit1.ControlNodes".fuses.E6480CB_vision_controller2_power_tripped )
      S_Coil( "Unit1.Alarms".systemFaultGeneral[64] )
   END_RUNG
   // the same network as SCL:
   IF NOT "Unit1.ControlNodes".fuses.E6480CB_vision_controller2_power_tripped THEN
       "Unit1.Alarms".systemFaultGeneral[64] := TRUE;
   END_IF;
END_REGION

REGION Network 73: PFE System Fault General 65
   RUNG wire#powerrail
      I_Contact( "Unit1.ControlNodes".fuses.E6486CB_vision_controller3_power_tripped )
      S_Coil( "Unit1.Alarms".systemFaultGeneral[65] )
   END_RUNG
   // the same network as SCL:
   IF NOT "Unit1.ControlNodes".fuses.E6486CB_vision_controller3_power_tripped THEN
       "Unit1.Alarms".systemFaultGeneral[65] := TRUE;
   END_IF;
END_REGION

REGION Network 74: PFE System Fault General 66
   RUNG wire#powerrail
      I_Contact( "Unit1.ControlNodes".fuses.E6506CB_linedLaser_module1_power_tripped )
      S_Coil( "Unit1.Alarms".systemFaultGeneral[66] )
   END_RUNG
   // the same network as SCL:
   IF NOT "Unit1.ControlNodes".fuses.E6506CB_linedLaser_module1_power_tripped THEN
       "Unit1.Alarms".systemFaultGeneral[66] := TRUE;
   END_IF;
END_REGION

REGION Network 75: PFE System Fault General 67
   RUNG wire#powerrail
      I_Contact( "Unit1.ControlNodes".fuses.E6512CB_linedLaser_module2_power_tripped )
      S_Coil( "Unit1.Alarms".systemFaultGeneral[67] )
   END_RUNG
   // the same network as SCL:
   IF NOT "Unit1.ControlNodes".fuses.E6512CB_linedLaser_module2_power_tripped THEN
       "Unit1.Alarms".systemFaultGeneral[67] := TRUE;
   END_IF;
END_REGION

REGION Network 76: PFE System Fault General 68
   RUNG wire#powerrail
      I_Contact( "Unit1.ControlNodes".fuses.E6706CB_controlLER_DC_power_tripped )
      S_Coil( "Unit1.Alarms".systemFaultGeneral[68] )
   END_RUNG
   // the same network as SCL:
   IF NOT "Unit1.ControlNodes".fuses.E6706CB_controlLER_DC_power_tripped THEN
       "Unit1.Alarms".systemFaultGeneral[68] := TRUE;
   END_IF;
END_REGION

REGION Network 77: PFE System Fault General 69
   RUNG wire#powerrail
      I_Contact( "Unit1.ControlNodes".fuses.E6716CB_EPC_controller1_power_tripped )
      S_Coil( "Unit1.Alarms".systemFaultGeneral[69] )
   END_RUNG
   // the same network as SCL:
   IF NOT "Unit1.ControlNodes".fuses.E6716CB_EPC_controller1_power_tripped THEN
       "Unit1.Alarms".systemFaultGeneral[69] := TRUE;
   END_IF;
END_REGION

REGION Network 78: PFE System Fault General 70
   RUNG wire#powerrail
      I_Contact( "Unit1.ControlNodes".fuses.E6722CB_EPC_controller2_power_tripped )
      S_Coil( "Unit1.Alarms".systemFaultGeneral[70] )
   END_RUNG
   // the same network as SCL:
   IF NOT "Unit1.ControlNodes".fuses.E6722CB_EPC_controller2_power_tripped THEN
       "Unit1.Alarms".systemFaultGeneral[70] := TRUE;
   END_IF;
END_REGION

REGION Network 79: PFE System Fault General 71
   RUNG wire#powerrail
      I_Contact( "Unit1.ControlNodes".fuses.E6728CB_EPC_controller3_power_tripped )
      S_Coil( "Unit1.Alarms".systemFaultGeneral[71] )
   END_RUNG
   // the same network as SCL:
   IF NOT "Unit1.ControlNodes".fuses.E6728CB_EPC_controller3_power_tripped THEN
       "Unit1.Alarms".systemFaultGeneral[71] := TRUE;
   END_IF;
END_REGION

REGION Network 80: PFE System Fault General 72
   RUNG wire#powerrail
      I_Contact( "Unit1.ControlNodes".fuses.E6734CB_EPC_controller4_power_tripped )
      S_Coil( "Unit1.Alarms".systemFaultGeneral[72] )
   END_RUNG
   // the same network as SCL:
   IF NOT "Unit1.ControlNodes".fuses.E6734CB_EPC_controller4_power_tripped THEN
       "Unit1.Alarms".systemFaultGeneral[72] := TRUE;
   END_IF;
END_REGION

REGION Network 81: PFE System Fault General 73
   RUNG wire#powerrail
      I_Contact( "Unit1.ControlNodes".fuses.E6806CB_safetyDc_power_tripped )
      S_Coil( "Unit1.Alarms".systemFaultGeneral[73] )
   END_RUNG
   // the same network as SCL:
   IF NOT "Unit1.ControlNodes".fuses.E6806CB_safetyDc_power_tripped THEN
       "Unit1.Alarms".systemFaultGeneral[73] := TRUE;
   END_IF;
END_REGION

REGION Network 82: PFE System Fault General 74
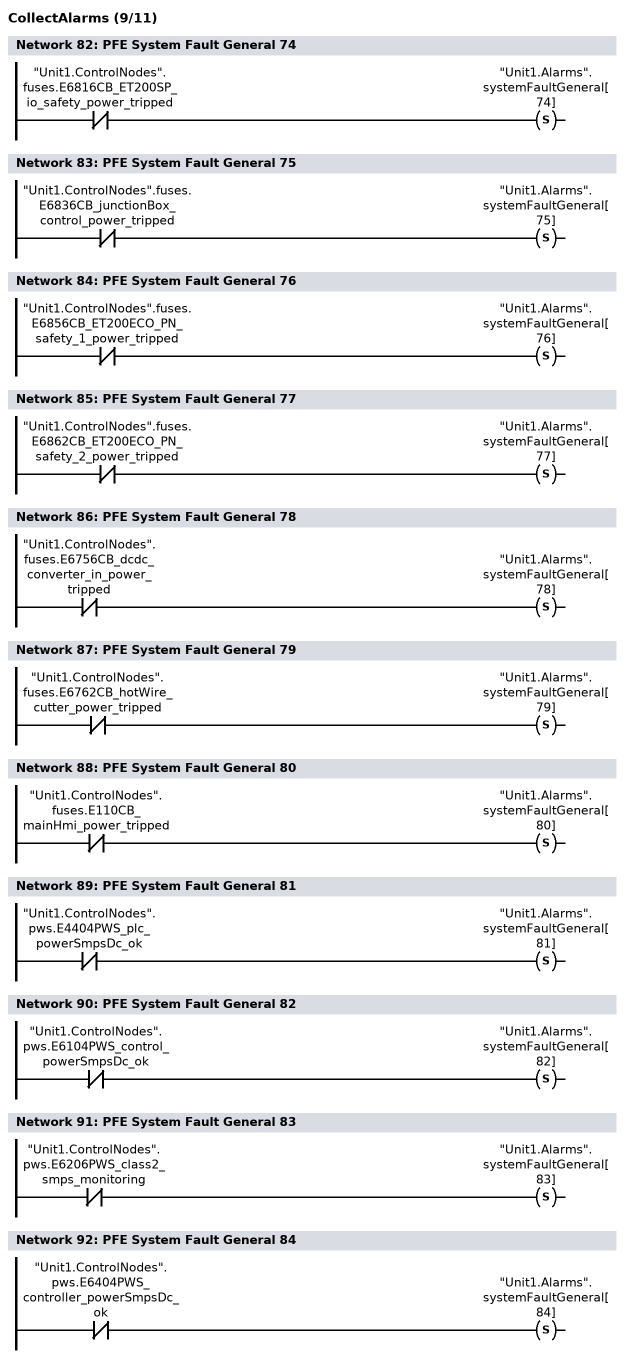
   RUNG wire#powerrail
      I_Contact( "Unit1.ControlNodes".fuses.E6816CB_ET200SP_io_safety_power_tripped )
      S_Coil( "Unit1.Alarms".systemFaultGeneral[74] )
   END_RUNG
   // the same network as SCL:
   IF NOT "Unit1.ControlNodes".fuses.E6816CB_ET200SP_io_safety_power_tripped THEN
       "Unit1.Alarms".systemFaultGeneral[74] := TRUE;
   END_IF;
END_REGION

REGION Network 83: PFE System Fault General 75
   RUNG wire#powerrail
      I_Contact( "Unit1.ControlNodes".fuses.E6836CB_junctionBox_control_power_tripped )
      S_Coil( "Unit1.Alarms".systemFaultGeneral[75] )
   END_RUNG
   // the same network as SCL:
   IF NOT "Unit1.ControlNodes".fuses.E6836CB_junctionBox_control_power_tripped THEN
       "Unit1.Alarms".systemFaultGeneral[75] := TRUE;
   END_IF;
END_REGION

REGION Network 84: PFE System Fault General 76
   RUNG wire#powerrail
      I_Contact( "Unit1.ControlNodes".fuses.E6856CB_ET200ECO_PN_safety_1_power_tripped )
      S_Coil( "Unit1.Alarms".systemFaultGeneral[76] )
   END_RUNG
   // the same network as SCL:
   IF NOT "Unit1.ControlNodes".fuses.E6856CB_ET200ECO_PN_safety_1_power_tripped THEN
       "Unit1.Alarms".systemFaultGeneral[76] := TRUE;
   END_IF;
END_REGION

REGION Network 85: PFE System Fault General 77
   RUNG wire#powerrail
      I_Contact( "Unit1.ControlNodes".fuses.E6862CB_ET200ECO_PN_safety_2_power_tripped )
      S_Coil( "Unit1.Alarms".systemFaultGeneral[77] )
   END_RUNG
   // the same network as SCL:
   IF NOT "Unit1.ControlNodes".fuses.E6862CB_ET200ECO_PN_safety_2_power_tripped THEN
       "Unit1.Alarms".systemFaultGeneral[77] := TRUE;
   END_IF;
END_REGION

REGION Network 86: PFE System Fault General 78
   RUNG wire#powerrail
      I_Contact( "Unit1.ControlNodes".fuses.E6756CB_dcdc_converter_in_power_tripped )
      S_Coil( "Unit1.Alarms".systemFaultGeneral[78] )
   END_RUNG
   // the same network as SCL:
   IF NOT "Unit1.ControlNodes".fuses.E6756CB_dcdc_converter_in_power_tripped THEN
       "Unit1.Alarms".systemFaultGeneral[78] := TRUE;
   END_IF;
END_REGION

REGION Network 87: PFE System Fault General 79
   RUNG wire#powerrail
      I_Contact( "Unit1.ControlNodes".fuses.E6762CB_hotWire_cutter_power_tripped )
      S_Coil( "Unit1.Alarms".systemFaultGeneral[79] )
   END_RUNG
   // the same network as SCL:
   IF NOT "Unit1.ControlNodes".fuses.E6762CB_hotWire_cutter_power_tripped THEN
       "Unit1.Alarms".systemFaultGeneral[79] := TRUE;
   END_IF;
END_REGION

REGION Network 88: PFE System Fault General 80
   RUNG wire#powerrail
      I_Contact( "Unit1.ControlNodes".fuses.E110CB_mainHmi_power_tripped )
      S_Coil( "Unit1.Alarms".systemFaultGeneral[80] )
   END_RUNG
   // the same network as SCL:
   IF NOT "Unit1.ControlNodes".fuses.E110CB_mainHmi_power_tripped THEN
       "Unit1.Alarms".systemFaultGeneral[80] := TRUE;
   END_IF;
END_REGION

REGION Network 89: PFE System Fault General 81
   RUNG wire#powerrail
      I_Contact( "Unit1.ControlNodes".pws.E4404PWS_plc_powerSmpsDc_ok )
      S_Coil( "Unit1.Alarms".systemFaultGeneral[81] )
   END_RUNG
   // the same network as SCL:
   IF NOT "Unit1.ControlNodes".pws.E4404PWS_plc_powerSmpsDc_ok THEN
       "Unit1.Alarms".systemFaultGeneral[81] := TRUE;
   END_IF;
END_REGION

REGION Network 90: PFE System Fault General 82
   RUNG wire#powerrail
      I_Contact( "Unit1.ControlNodes".pws.E6104PWS_control_powerSmpsDc_ok )
      S_Coil( "Unit1.Alarms".systemFaultGeneral[82] )
   END_RUNG
   // the same network as SCL:
   IF NOT "Unit1.ControlNodes".pws.E6104PWS_control_powerSmpsDc_ok THEN
       "Unit1.Alarms".systemFaultGeneral[82] := TRUE;
   END_IF;
END_REGION

REGION Network 91: PFE System Fault General 83
   RUNG wire#powerrail
      I_Contact( "Unit1.ControlNodes".pws.E6206PWS_class2_smps_monitoring )
      S_Coil( "Unit1.Alarms".systemFaultGeneral[83] )
   END_RUNG
   // the same network as SCL:
   IF NOT "Unit1.ControlNodes".pws.E6206PWS_class2_smps_monitoring THEN
       "Unit1.Alarms".systemFaultGeneral[83] := TRUE;
   END_IF;
END_REGION

REGION Network 92: PFE System Fault General 84
   RUNG wire#powerrail
      I_Contact( "Unit1.ControlNodes".pws.E6404PWS_controller_powerSmpsDc_ok )
      S_Coil( "Unit1.Alarms".systemFaultGeneral[84] )
   END_RUNG
   // the same network as SCL:
   IF NOT "Unit1.ControlNodes".pws.E6404PWS_controller_powerSmpsDc_ok THEN
       "Unit1.Alarms".systemFaultGeneral[84] := TRUE;
   END_IF;
END_REGION

REGION Network 93: PFE System Fault General 85
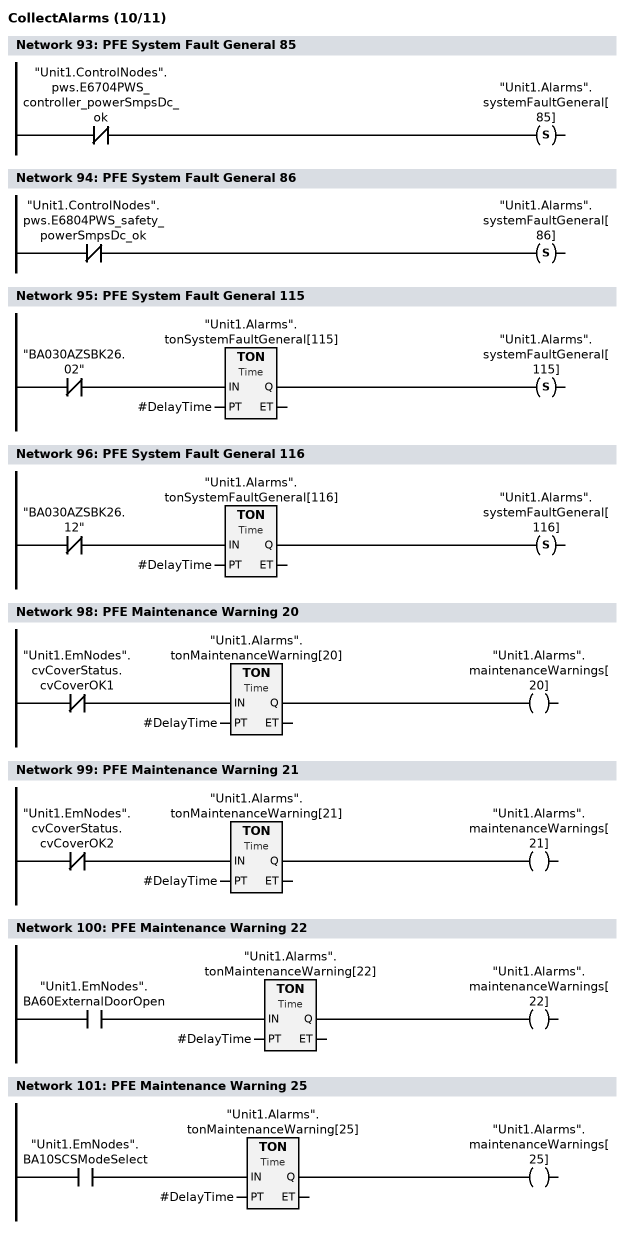
   RUNG wire#powerrail
      I_Contact( "Unit1.ControlNodes".pws.E6704PWS_controller_powerSmpsDc_ok )
      S_Coil( "Unit1.Alarms".systemFaultGeneral[85] )
   END_RUNG
   // the same network as SCL:
   IF NOT "Unit1.ControlNodes".pws.E6704PWS_controller_powerSmpsDc_ok THEN
       "Unit1.Alarms".systemFaultGeneral[85] := TRUE;
   END_IF;
END_REGION

REGION Network 94: PFE System Fault General 86
   RUNG wire#powerrail
      I_Contact( "Unit1.ControlNodes".pws.E6804PWS_safety_powerSmpsDc_ok )
      S_Coil( "Unit1.Alarms".systemFaultGeneral[86] )
   END_RUNG
   // the same network as SCL:
   IF NOT "Unit1.ControlNodes".pws.E6804PWS_safety_powerSmpsDc_ok THEN
       "Unit1.Alarms".systemFaultGeneral[86] := TRUE;
   END_IF;
END_REGION

REGION Network 95: PFE System Fault General 115
   RUNG wire#powerrail
      I_Contact( "BA030AZSBK26.02" )
      { S7_Templates := "time_type := Time" } "Unit1.Alarms".tonSystemFaultGeneral[115].TON(pt := #DelayTime, et =>)
      S_Coil( "Unit1.Alarms".systemFaultGeneral[115] )
   END_RUNG
   // the same network as SCL:
   "Unit1.Alarms".tonSystemFaultGeneral[115].TON(IN := NOT "BA030AZSBK26.02", PT := #DelayTime);
   IF "Unit1.Alarms".tonSystemFaultGeneral[115].Q THEN
       "Unit1.Alarms".systemFaultGeneral[115] := TRUE;
   END_IF;
END_REGION

REGION Network 96: PFE System Fault General 116
   RUNG wire#powerrail
      I_Contact( "BA030AZSBK26.12" )
      { S7_Templates := "time_type := Time" } "Unit1.Alarms".tonSystemFaultGeneral[116].TON(pt := #DelayTime, et =>)
      S_Coil( "Unit1.Alarms".systemFaultGeneral[116] )
   END_RUNG
   // the same network as SCL:
   "Unit1.Alarms".tonSystemFaultGeneral[116].TON(IN := NOT "BA030AZSBK26.12", PT := #DelayTime);
   IF "Unit1.Alarms".tonSystemFaultGeneral[116].Q THEN
       "Unit1.Alarms".systemFaultGeneral[116] := TRUE;
   END_IF;
END_REGION

REGION Network 97: *************** Warning **************************
END_REGION

REGION Network 98: PFE Maintenance Warning 20
   RUNG wire#powerrail
      I_Contact( "Unit1.EmNodes".cvCoverStatus.cvCoverOK1 )
      { S7_Templates := "time_type := Time" } "Unit1.Alarms".tonMaintenanceWarning[20].TON(pt := #DelayTime, et =>)
      Coil( "Unit1.Alarms".maintenanceWarnings[20] )
   END_RUNG
   // the same network as SCL:
   "Unit1.Alarms".tonMaintenanceWarning[20].TON(IN := NOT "Unit1.EmNodes".cvCoverStatus.cvCoverOK1,
                           PT := #DelayTime);
   "Unit1.Alarms".maintenanceWarnings[20] := "Unit1.Alarms".tonMaintenanceWarning[20].Q;
END_REGION

REGION Network 99: PFE Maintenance Warning 21
   RUNG wire#powerrail
      I_Contact( "Unit1.EmNodes".cvCoverStatus.cvCoverOK2 )
      { S7_Templates := "time_type := Time" } "Unit1.Alarms".tonMaintenanceWarning[21].TON(pt := #DelayTime, et =>)
      Coil( "Unit1.Alarms".maintenanceWarnings[21] )
   END_RUNG
   // the same network as SCL:
   "Unit1.Alarms".tonMaintenanceWarning[21].TON(IN := NOT "Unit1.EmNodes".cvCoverStatus.cvCoverOK2,
                           PT := #DelayTime);
   "Unit1.Alarms".maintenanceWarnings[21] := "Unit1.Alarms".tonMaintenanceWarning[21].Q;
END_REGION

REGION Network 100: PFE Maintenance Warning 22
   RUNG wire#powerrail
      Contact( "Unit1.EmNodes".BA60ExternalDoorOpen )
      { S7_Templates := "time_type := Time" } "Unit1.Alarms".tonMaintenanceWarning[22].TON(pt := #DelayTime, et =>)
      Coil( "Unit1.Alarms".maintenanceWarnings[22] )
   END_RUNG
   // the same network as SCL:
   "Unit1.Alarms".tonMaintenanceWarning[22].TON(IN := "Unit1.EmNodes".BA60ExternalDoorOpen, PT := #DelayTime);
   "Unit1.Alarms".maintenanceWarnings[22] := "Unit1.Alarms".tonMaintenanceWarning[22].Q;
END_REGION

REGION Network 101: PFE Maintenance Warning 25
   RUNG wire#powerrail
      Contact( "Unit1.EmNodes".BA10SCSModeSelect )
      { S7_Templates := "time_type := Time" } "Unit1.Alarms".tonMaintenanceWarning[25].TON(pt := #DelayTime, et =>)
      Coil( "Unit1.Alarms".maintenanceWarnings[25] )
   END_RUNG
   // the same network as SCL:
   "Unit1.Alarms".tonMaintenanceWarning[25].TON(IN := "Unit1.EmNodes".BA10SCSModeSelect, PT := #DelayTime);
   "Unit1.Alarms".maintenanceWarnings[25] := "Unit1.Alarms".tonMaintenanceWarning[25].Q;
END_REGION

REGION Network 102: PFE Maintenance Warning 26
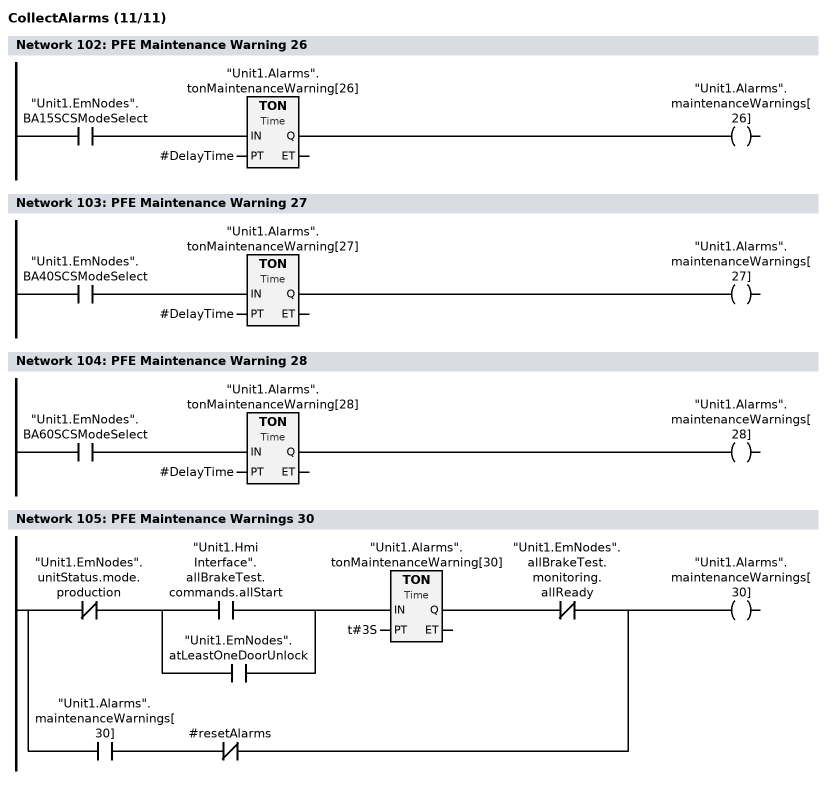
   RUNG wire#powerrail
      Contact( "Unit1.EmNodes".BA15SCSModeSelect )
      { S7_Templates := "time_type := Time" } "Unit1.Alarms".tonMaintenanceWarning[26].TON(pt := #DelayTime, et =>)
      Coil( "Unit1.Alarms".maintenanceWarnings[26] )
   END_RUNG
   // the same network as SCL:
   "Unit1.Alarms".tonMaintenanceWarning[26].TON(IN := "Unit1.EmNodes".BA15SCSModeSelect, PT := #DelayTime);
   "Unit1.Alarms".maintenanceWarnings[26] := "Unit1.Alarms".tonMaintenanceWarning[26].Q;
END_REGION

REGION Network 103: PFE Maintenance Warning 27
   RUNG wire#powerrail
      Contact( "Unit1.EmNodes".BA40SCSModeSelect )
      { S7_Templates := "time_type := Time" } "Unit1.Alarms".tonMaintenanceWarning[27].TON(pt := #DelayTime, et =>)
      Coil( "Unit1.Alarms".maintenanceWarnings[27] )
   END_RUNG
   // the same network as SCL:
   "Unit1.Alarms".tonMaintenanceWarning[27].TON(IN := "Unit1.EmNodes".BA40SCSModeSelect, PT := #DelayTime);
   "Unit1.Alarms".maintenanceWarnings[27] := "Unit1.Alarms".tonMaintenanceWarning[27].Q;
END_REGION

REGION Network 104: PFE Maintenance Warning 28
   RUNG wire#powerrail
      Contact( "Unit1.EmNodes".BA60SCSModeSelect )
      { S7_Templates := "time_type := Time" } "Unit1.Alarms".tonMaintenanceWarning[28].TON(pt := #DelayTime, et =>)
      Coil( "Unit1.Alarms".maintenanceWarnings[28] )
   END_RUNG
   // the same network as SCL:
   "Unit1.Alarms".tonMaintenanceWarning[28].TON(IN := "Unit1.EmNodes".BA60SCSModeSelect, PT := #DelayTime);
   "Unit1.Alarms".maintenanceWarnings[28] := "Unit1.Alarms".tonMaintenanceWarning[28].Q;
END_REGION

REGION Network 105: PFE Maintenance Warnings 30
   RUNG wire#powerrail
      I_Contact( "Unit1.EmNodes".unitStatus.mode.production )
      wire#w1
      Contact( "Unit1.HmiInterface".allBrakeTest.commands.allStart )
      wire#w2
      { S7_Templates := "time_type := Time" } "Unit1.Alarms".tonMaintenanceWarning[30].TON(pt := t#3S, et =>)
      I_Contact( "Unit1.EmNodes".allBrakeTest.monitoring.allReady )
      wire#w3
      Coil( "Unit1.Alarms".maintenanceWarnings[30] )
   END_RUNG
   RUNG wire#w1
      Contact( "Unit1.EmNodes".atLeastOneDoorUnlock )
   END_RUNG wire#w2
   RUNG wire#powerrail
      Contact( "Unit1.Alarms".maintenanceWarnings[30] )
      I_Contact( #resetAlarms )
   END_RUNG wire#w3
   // the same network as SCL:
   "Unit1.Alarms".tonMaintenanceWarning[30].TON(IN := NOT "Unit1.EmNodes".unitStatus.mode.production AND ("Unit1.HmiInterface".allBrakeTest.commands.allStart OR "Unit1.EmNodes".atLeastOneDoorUnlock),
                           PT := t#3S);
   "Unit1.Alarms".maintenanceWarnings[30] := ("Unit1.Alarms".tonMaintenanceWarning[30].Q AND NOT "Unit1.EmNodes".allBrakeTest.monitoring.allReady) OR ("Unit1.Alarms".maintenanceWarnings[30] AND NOT #resetAlarms);
END_REGION
END_FUNCTION
